Omron Sysmac Studio project ExampleControlWithAIShell (Sysmac Studio 1.63.0.7, StandardProject)

# Controller Example: NX102-9000 version 1.64
Units and slaves: ユニット1 : NX-PF0630(N1); ユニット2 : NX-ID4442(N2); ユニット3 : NX-ID4442(N3); ユニット4 : NX-OD4256(N4); ユニット5 : NX-OD4256(N5); ユニット6 : NX-AD2603(N6)
Axis MC_Axis1, settings changed from default: AxisType=ServoType, FunctionLimit=SingleAxisPTP, UnitsConversion=EnumElement2, UnitsNumerator=8388608, UnitsDenominator=10, TravelDistancePerWorkRotation=5, MaxVelocity=200, MaxJogVelocity=200, InPositionBand=1, ZeroPositionBand=1, FollowingErrorLimit=5, FollowingErrorAlarmLimit=1, EncoderTypes=Abs
Axis MC_Axis2, settings changed from default: AxisNumber=1, AxisType=ServoType, FunctionLimit=SingleAxisPTP, UnitsConversion=EnumElement5, UnitsNumerator=8388608, UnitsDenominator=360, MaxVelocity=36000, MaxJogVelocity=36000, InPositionBand=0.1, ModuloMAXPosition=360, ModuloMINPosition=0
Task PrimaryTask (priority 4, period or condition 2000): Main, SimDriveReflection, DeviceInterfaces
Library UAMotionLinkLib 0.0.1 (contents left out)

TYPE SliderModel : STRUCT
    CtrlImmediateStop : BOOL;
    CtrlStop : BOOL;
    CtrlServoOn : BOOL;
    CtrlResetError : BOOL;
    CtrlJogLeft : BOOL;
    CtrlJogRight : BOOL;
    CtrlMoveToZero : BOOL;
    CtrlHome : BOOL;
    AllowMotion : BOOL;
    PowerOn : BOOL;
    NegLimit : BOOL;
    PosLimit : BOOL;
    Velocity : REAL;
END_STRUCT END_TYPE



PROGRAM README
RETURN;
(*
This project is related to the following:

https://github.com/kmu2030/UAMotionLinkLib/examples/ControlWithAIShell


このプロジェクトは、以下に関連したプロジェクトです。

https://github.com/kmu2030/UAMotionLinkLib/examples/ControlWithAIShell

For the parts to which I have rights, I follow POU/PROGRAM/LICENSE.
You are free to use and modify it, but we are not responsible for any damage or loss related to it.
*)
END_PROGRAM

PROGRAM LICENSE
RETURN;
(*
The MIT License (MIT)

Copyright(c) 2025 KITA Munemitsu

Permission is hereby granted, free of charge, to any person obtaining a copy of this software and associated
documentation files (the “Software”), to deal in the Software without restriction, including without limitation
the rights to use, copy, modify, merge, publish, distribute, sublicense, and/or sell copies of the Software,
and to permit persons to whom the Software is furnished to do so, subject to the following conditions:

The above copyright notice and this permission notice shall be included in all copies or substantial portions of the Software.

THE SOFTWARE IS PROVIDED “AS IS”, WITHOUT WARRANTY OF ANY KIND, EXPRESS OR IMPLIED, INCLUDING BUT NOT
LIMITED TO THE WARRANTIES OF MERCHANTABILITY, FITNESS FOR A PARTICULAR PURPOSE AND NONINFRINGEMENT.
IN NO EVENT SHALL THE AUTHORS OR COPYRIGHT HOLDERS BE LIABLE FOR ANY CLAIM, DAMAGES OR OTHER LIABILITY,
WHETHER IN AN ACTION OF CONTRACT, TORT OR OTHERWISE, ARISING FROM, OUT OF OR IN CONNECTION WITH THE SOFTWARE
OR THE USE OR OTHER DEALINGS IN THE SOFTWARE.
*)
END_PROGRAM

PROGRAM Main
VAR
    iSliderController : SliderController;
    iSliderModel : SliderModel;
END_VAR
VAR_EXTERNAL CONSTANT
    _MC_AX : ARRAY[0..15] OF _sAXIS_REF;
END_VAR
IF P_First_Run THEN
	iSliderModel.CtrlServoOn := TRUE;
	iSliderModel.CtrlStop := FALSE;
	iSliderModel.CtrlImmediateStop := FALSE;
	iSliderModel.CtrlMoveToZero := FALSE;
	iSliderModel.CtrlJogLeft := FALSE;
	iSliderModel.CtrlJogRight := FALSE;
	iSliderModel.CtrlHome := FALSE;
	iSliderModel.CtrlResetError := FALSE;
	
	iSliderController.Enable := TRUE;
END_IF;

// Signals
iSliderModel.PowerOn := TRUE;
iSliderModel.PosLimit := FALSE;
iSliderModel.NegLimit := FALSE;
iSliderModel.AllowMotion := TRUE;

iSliderController(Axis:=_MC_AX[0],
				  Model:=iSliderModel);
END_PROGRAM

PROGRAM SimDriveReflection
VAR
    iSimMCRefrectors : ARRAY[0..15] OF SimMCReflector;
    i : UINT;
END_VAR
VAR_EXTERNAL CONSTANT
    _MC_AX : ARRAY[0..15] OF _sAXIS_REF;
END_VAR
IF P_First_Run THEN
	iSimMCRefrectors[0].Enable := TRUE;
	iSimMCRefrectors[1].Enable := TRUE;
END_IF;

// Simulation
FOR i := 0 TO 15 DO
	iSimMCRefrectors[i](Axis:=_MC_AX[i]);
END_FOR;
END_PROGRAM

PROGRAM DeviceInterfaces
VAR
    SingleMCController : BasicMCControllerModel;
END_VAR
VAR_EXTERNAL CONSTANT
    _MC_AX : ARRAY[0..15] OF _sAXIS_REF;
END_VAR
IF P_First_Run THEN
	SingleMCController.Enable := TRUE;
	SingleMCController.AllowControl := TRUE;
END_IF;

SingleMCController(Axes:=_MC_AX);
END_PROGRAM

FUNCTION_BLOCK SliderController
VAR
    iMC_ImmediateStop : MC_ImmediateStop;
    iMC_Stop : MC_Stop;
    iMC_Power : MC_Power;
    iMC_Reset : MC_Reset;
    iMC_Home : MC_Home;
    iMC_MoveJog : MC_MoveJog;
    iMC_MoveZeroPosition : MC_MoveZeroPosition;
END_VAR
VAR CONSTANT
    STATE_INIT : UINT := 0;
    STATE_WAIT : UINT := 10;
    STATE_JOG_LEFT : UINT := 20;
    STATE_JOG_RIGHT : UINT := 30;
    STATE_MOVE_TO_ZERO : UINT := 40;
    STATE_HOME : UINT := 70;
    STATE_STOP : UINT := 80;
    STATE_RESET_ERROR : UINT := 90;
    STATE_IMMEDIATE_STOP : UINT := 100;
    STATE_DONE : UINT := 1000;
END_VAR
VAR
    iState : UINT := 1001;
    iStop : BOOL;
    iPrevStop : BOOL;
END_VAR
VAR_INPUT
    Enable : BOOL;
END_VAR
VAR_IN_OUT CONSTANT
    Axis : _sAXIS_REF;
END_VAR
VAR_IN_OUT
    Model : SliderModel;
END_VAR
VAR_OUTPUT
    Busy : BOOL;
END_VAR
IF Enable AND NOT Busy THEN
	Busy := TRUE;
	
	iState := STATE_INIT;
END_IF;

iPrevStop := iStop;
iStop := Model.CtrlStop
	OR iMC_Power.Error
	OR NOT Model.AllowMotion;

IF Model.CtrlImmediateStop THEN
	iState := STATE_IMMEDIATE_STOP;
ELSIF iStop AND NOT iPrevStop THEN
	CASE iState OF
		20..69:
			iMC_MoveJog.NegativeEnable := FALSE;
			iMC_MoveJog.PositiveEnable := FALSE;
			iMC_MoveZeroPosition.Execute := FALSE;
			
			iState := STATE_STOP;
	END_CASE;
END_IF;

CASE iState OF
	// STATE_INIT
	0:
		iMC_ImmediateStop.Execute := FALSE;
		iMC_Stop.Execute := FALSE;
		iMC_Power.Enable := FALSE;
		iMC_Reset.Execute := FALSE;
		iMC_Home.Execute := FALSE;
		iMC_MoveJog.NegativeEnable := FALSE;
		iMC_MoveJog.PositiveEnable := FALSE;
		iMC_MoveZeroPosition.Execute := FALSE;
		
		IF NOT Enable THEN
			iState := STATE_DONE;
		ELSE
			Inc(iState);
		END_IF;
	1:
		IF Model.PowerOn THEN
			Inc(iState);
		END_IF;
	2:
		IF Model.CtrlServoOn THEN
			iMC_Power.Enable := TRUE;
			
			Inc(iState);
		END_IF;
	3:
		IF Axis.DrvStatus.ServoOn THEN
			iState := STATE_WAIT;
		ELSIF iMC_Power.Error THEN
			iState := STATE_INIT;
		END_IF;

	// STATE_WAIT
	10:
		IF NOT Model.PowerOn
			OR NOT Model.CtrlServoOn
			OR iMC_Power.Error
		THEN
			iMC_Power.Enable := FALSE;
			
			iState := STATE_INIT;			
		ELSIF Model.CtrlStop THEN
			iState := STATE_STOP;
		ELSIF Model.CtrlResetError THEN
			iState := STATE_RESET_ERROR;
		ELSIF Model.CtrlHome THEN
			iState := STATE_HOME;
		ELSIF Model.AllowMotion THEN
			IF Model.CtrlJogLeft THEN
				iState := STATE_JOG_LEFT;
			ELSIF Model.CtrlJogRight THEN
				iState := STATE_JOG_RIGHT;
			ELSIF Model.CtrlMoveToZero THEN
				iState := STATE_MOVE_TO_ZERO;
			END_IF;
		END_IF;

	// STATE_JOG_LFET
	20:
		IF Model.NegLimit THEN
			iState := iState + 9;
		ELSIF Model.CtrlJogLeft THEN
			iMC_MoveJog.NegativeEnable := TRUE;
			iMC_MoveJog.Velocity := Model.Velocity;
			
			Inc(iState);
		END_IF;
	21:
		IF iMC_MoveJog.Error THEN
			iMC_MoveJog.NegativeEnable := FALSE;
			iMC_Stop.Execute := TRUE;
			
			Inc(iState);
		ELSIF NOT Model.CtrlJogLeft OR Model.NegLimit THEN
			iMC_MoveJog.NegativeEnable := FALSE;
			iMC_Stop.Execute := TRUE;
					
			Inc(iState);
		END_IF;
	22:
		IF iMC_Stop.Done OR iMC_Stop.Error THEN
			iMC_Stop.Execute := FALSE;
			
			iState := iState + 7;
		END_IF;
	29:
		IF Axis.Status.Standstill THEN
			iState := STATE_WAIT;
		END_IF;

	// STATE_JOG_RIGHT
	30:
		IF Model.PosLimit THEN
			iState := iState + 9;
		ELSIF Model.CtrlJogRight THEN
			iMC_MoveJog.PositiveEnable := TRUE;
			iMC_MoveJog.Velocity := Model.Velocity;
			
			Inc(iState);
		END_IF;
	31:
		IF iMC_MoveJog.Error THEN
			iMC_MoveJog.PositiveEnable := FALSE;
			iMC_Stop.Execute := TRUE;
			
			Inc(iState);
		ELSIF NOT Model.CtrlJogRight OR Model.PosLimit THEN
			iMC_MoveJog.PositiveEnable := FALSE;
			iMC_Stop.Execute := TRUE;
					
			Inc(iState);
		END_IF;
	32:
		IF iMC_Stop.Done OR iMC_Stop.Error THEN
			iMC_Stop.Execute := FALSE;
			
			iState := iState + 7;
		END_IF;
	39:
		IF Axis.Status.Standstill THEN
			iState := STATE_WAIT;
		END_IF;
	
	// STATE_MOVE_TO_ZERO
	40:
		iMC_MoveZeroPosition.Velocity := Model.Velocity;
		iMC_MoveZeroPosition.Execute := TRUE;
		
		Inc(iState);
	41:
		IF iMC_MoveZeroPosition.Done OR iMC_MoveZeroPosition.Error THEN
			iMC_MoveZeroPosition.Execute := FALSE;
			
			iState := iState + 8;
		END_IF;
	49:
		IF NOT Model.CtrlMoveToZero THEN
			iState := STATE_WAIT;
		END_IF;

	// STATE_HOME
	70:
		iMC_Home.Execute := TRUE;
		
		Inc(iState);
	71:
		IF iMC_Home.Done OR iMC_Home.Error THEN
			iMC_Home.Execute := FALSE;
			
			iState := iState + 8;
		END_IF;
	79:
		IF NOT Model.CtrlHome THEN
			iState := STATE_WAIT;
		END_IF;

	// STATE_STOP
	80:
		iMC_MoveJog.NegativeEnable := FALSE;
		iMC_MoveJog.PositiveEnable := FALSE;
		iMC_MoveZeroPosition.Execute := FALSE;
		
		IF Axis.Status.Standstill THEN
			iState := iState + 9;
		ELSE
			iMC_Stop.BufferMode := _eMC_BUFFER_MODE#_mcAborting;
			iMC_Stop.Execute := TRUE;
		
			Inc(iState);
		END_IF;
	81:
		IF iMC_Stop.Done OR iMC_Stop.Error THEN
			iMC_Stop.Execute := FALSE;
			
			iState := iState + 8;
		END_IF;
	89:
		IF Axis.Status.Standstill THEN
			iState := STATE_WAIT;
		END_IF;

	// STATE_RESET_ERROR
	90:
		iMC_Reset.Execute := TRUE;
		
		Inc(iState);
	91:
		IF iMC_Reset.Done OR iMC_Reset.Error THEN
			iMC_Reset.Execute := FALSE;
			
			iState := iState + 8;
		END_IF;
	99:
		IF NOT Model.CtrlResetError THEN
			iState := STATE_WAIT;
		END_IF;
		
	// STATE_IMMADIATE_STOP
	100:
		iMC_MoveJog.PositiveEnable := FALSE;
		iMC_MoveJog.NegativeEnable := FALSE;
		iMC_MoveZeroPosition.Execute := FALSE;

		iMC_ImmediateStop.StopMode := _eMC_STOP_MODE#_mcImmediateStop;
		iMC_ImmediateStop.Execute := TRUE;
		
		Inc(iState);
	101:
		IF iMC_ImmediateStop.Done OR iMC_ImmediateStop.Error THEN
			iMC_ImmediateStop.Execute := FALSE;
			
			iState := iState + 8;
		END_IF;
	109:
		IF NOT Model.CtrlImmediateStop THEN
			iState := STATE_WAIT;
		END_IF;
	
	// STATE_DONE
	1000:
		Busy := FALSE;
		
		Inc(iState);
END_CASE;

iMC_ImmediateStop(Axis:=Axis);
iMC_Stop(Axis:=Axis);
iMC_Power(Axis:=Axis);
iMC_Reset(Axis:=Axis);
iMC_Home(Axis:=Axis);
iMC_MoveJog(Axis:=Axis);
iMC_MoveZeroPosition(Axis:=Axis);
END_FUNCTION_BLOCK

FUNCTION_BLOCK SimMCReflector
VAR
    iSimSetActPos : SIM_SetActPos;
    iSimSetActVel : SIM_SetActVel;
    iSimSetActTrq : SIM_SetActTrq;
    iSimSigNegLim : SIM_SigNegLmt;
    iSimSigPosLim : SIM_SigPosLmt;
END_VAR
VAR CONSTANT
    STATE_INIT : UINT := 0;
    STATE_WAIT : UINT := 10;
    STATE_REFRECT_MOTION : UINT := 20;
    STATE_DONE : UINT := 1000;
END_VAR
VAR
    iState : UINT := 1001;
END_VAR
VAR_INPUT
    Enable : BOOL;
END_VAR
VAR_IN_OUT CONSTANT
    Axis : _sAXIS_REF;
END_VAR
VAR_OUTPUT
    Busy : BOOL;
END_VAR
CASE Axis.Cfg.AxEnable OF
	_eMC_AXIS_USE#_mcNoneAxis,
	_eMC_AXIS_USE#_mcUnusedAxis:
		RETURN;
END_CASE;

IF Enable AND NOT Busy THEN
	Busy := TRUE;
	
	iState := STATE_INIT;
END_IF;

CASE iState OF
	// STATE_INIT
	0:
		iSimSetActPos.Enable := FALSE;
		iSimSetActVel.Enable := FALSE;
		iSimSetActTrq.Enable := FALSE;
		
		iState := STATE_WAIT;
	
	// STATE_WAIT
	10:
		IF NOT Enable THEN
			iState := STATE_DONE;
		ELSIF NOT Axis.Status.Standstill THEN
			iSimSetActPos.SetPos := Axis.Cmd.Pos;
			iSimSetActVel.SetVel := Axis.Cmd.Vel;
			iSimSetActTrq.SetTrq := Axis.Cmd.Trq;
			iSimSetActPos.Enable := TRUE;
			iSimSetActVel.Enable := TRUE;
			iSimSetActTrq.Enable := TRUE;

			iState := STATE_REFRECT_MOTION;
		END_IF;

	// STATE_REFRECT_MOTION
	20:
		iSimSetActPos.SetPos := Axis.Cmd.Pos;
		iSimSetActVel.SetVel := Axis.Cmd.Vel;
		iSimSetActTrq.SetTrq := Axis.Cmd.Trq;
		IF Axis.Status.Standstill THEN
			iState := iState + 9;
		END_IF;
	29:
		iSimSetActPos.Enable := FALSE;
		iSimSetActVel.Enable := FALSE;
		iSimSetActTrq.Enable := FALSE;
		
		iState := STATE_WAIT;
	
	// STATE_DONE
	1000:
		iSimSetActPos.Enable := FALSE;
		iSimSetActVel.Enable := FALSE;
		iSimSetActTrq.Enable := FALSE;
		
		Busy := FALSE;
		
		Inc(iState);
END_CASE;

iSimSetActPos(Axis:=Axis);
iSimSetActVel(Axis:=Axis);
iSimSetActTrq(Axis:=Axis);
END_FUNCTION_BLOCK